{attribute 'linkalways'} 
{attribute 'no_explicit_call' := 'This FB is a CLASS and must be accessed using methods or properties'}
{attribute 'enable_dynamic_creation'}
FUNCTION_BLOCK _ETcVnTimestamp EXTENDS EnumDatatypeBase
VAR
	localData : ETcVnTimestamp;
	activeData : REFERENCE TO ETcVnTimestamp;
	enumBaseDatatype : _ULINT(localData);
END_VAR

METHOD PRIVATE AddLocalEnumeration
VAR_INPUT
	Enumeration : T_MAXSTRING;
	Value : ETcVnTimestamp;
END_VAR
AddEnumeration(Enumeration, Value);
END_METHOD

PROPERTY PUBLIC Address : PVOID
GET
Address := ADR(activeData);
END_GET
END_PROPERTY

METHOD PUBLIC ClearReference
VAR_INPUT
END_VAR
activeData REF= localData;
SetBaseDatatypeReference();
END_METHOD

METHOD PUBLIC Clone : I_Datatype
VAR
    pClone : POINTER TO _ETcVnTimestamp;
END_VAR
pClone := __NEW(_ETcVnTimestamp(InitialValue := Value));
Clone := pClone^;
END_METHOD

METHOD FB_init : BOOL
VAR_INPUT
	bInitRetains : BOOL; // if TRUE, the retain variables are initialized (warm start / cold start)
	bInCopyCode : BOOL;  // if TRUE, the instance afterwards gets moved into the copy code (online change)
	InitialValue : ETcVnTimestamp;
END_VAR
localData := InitialValue;
AddBaseDatatype(enumBaseDatatype);
ClearReference();

AddLocalEnumeration('TCVN_TS_IMAGE_COMPLETED', ETcVnTimestamp.TCVN_TS_IMAGE_COMPLETED);
AddLocalEnumeration('TCVN_TS_RECEPTION_STARTED', ETcVnTimestamp.TCVN_TS_RECEPTION_STARTED);
AddLocalEnumeration('TCVN_TS_RECEPTION_FINISHED', ETcVnTimestamp.TCVN_TS_RECEPTION_FINISHED);
AddLocalEnumeration('TCVN_TS_GETCURRENTIMAGE', ETcVnTimestamp.TCVN_TS_GETCURRENTIMAGE);
AddLocalEnumeration('TCVN_TS_CAMERA', ETcVnTimestamp.TCVN_TS_CAMERA);
AddLocalEnumeration('TCVN_TS_CUSTOM', ETcVnTimestamp.TCVN_TS_CUSTOM);
AddLocalEnumeration('TCVN_TS_LAST_CHANGE', ETcVnTimestamp.TCVN_TS_LAST_CHANGE);
END_METHOD

PROPERTY PUBLIC Identifier : T_MAXSTRING
GET
Identifier := 'ETcVnTimestamp';
END_GET
END_PROPERTY

METHOD IsEnumeratorValueEqual : BOOL
VAR_INPUT
	Enumerator : I_KeyValueForwardEnumerator;
END_VAR
VAR
	storedValue : ETcVnTimestamp;
END_VAR
IF NOT Enumerator.TryGet(storedValue) THEN
	RETURN;
END_IF

IsEnumeratorValueEqual := storedValue = activeData;
END_METHOD

METHOD PUBLIC MakeReferenceTo
VAR_INPUT
	ReferenceTarget : REFERENCE TO ETcVnTimestamp;
END_VAR
activeData REF= ReferenceTarget;
SetBaseDatatypeReference();
END_METHOD

METHOD PROTECTED SetBaseDatatypeReference
VAR_INPUT
END_VAR
enumBaseDatatype.MakeReferenceTo(activeData);
END_METHOD

PROPERTY PUBLIC Size : UDINT
GET
Size := SIZEOF(activeData);
END_GET
END_PROPERTY

METHOD TryMakeReferenceTo : BOOL
VAR_INPUT
	Target : I_Datatype;
END_VAR
VAR
	pTargetData : POINTER TO ETcVnTimestamp;
END_VAR
IF NOT IsEquivalentTo(Target) THEN
	RETURN;
END_IF

pTargetData := Target.Address;
activeData REF= pTargetData^;
SetBaseDatatypeReference();
TryMakeReferenceTo := TRUE;
END_METHOD

PROPERTY PUBLIC Value : ETcVnTimestamp
GET
Value := activeData;
END_GET
SET
activeData := Value;
END_SET
END_PROPERTY

END_FUNCTION_BLOCK

(* stored: Version 1.1.0.1, ProductVersion 3.1.4024.13
   POU _ETcVnTimestamp: Id {d310adf1-2d37-00bd-1115-27d104ed3ef1}, SpecialFunc None
   Folder Core: Id {77af2560-cced-0daa-1211-123cfc3f2b65}
   Folder Protected: Id {f197ed99-828c-03bc-1837-1248521862bf}
   Folder Customize: Id {a26a2583-c016-0ec1-1b4d-be17805a6222}
   Folder Constructor: Id {2f2e0018-e3d4-06bb-102f-a67267979187}
   Folder Private: Id {c1d5397d-7f83-04fc-00f1-6b2625b52d99}
   Folder Protected: Id {52aaf5b4-eb11-0bc2-3716-f2f8b90090b1}
   Method AddLocalEnumeration: Id {77d22b0d-a8d9-0cc2-2753-4dd5ac642356}
   Property Address: Id {859ab322-5f62-0381-1503-fb6a93686b75}
   Get Get: Id {3d2bfc6b-7a64-08f3-1a17-af947191ef54}
   Method ClearReference: Id {95f88eef-d490-0511-0202-d3cf57e680b4}
   Method Clone: Id {daa1e185-a8b6-0b39-333e-ce61777f51c2}
   Method FB_init: Id {9f033ef3-530e-0765-08c7-8923a6e6ad97}
   Property Identifier: Id {06515588-f3ce-01c0-170e-fa8c1bf802a9}
   Get Get: Id {703d6092-be97-00bd-3087-38ab1f5f081f}
   Method IsEnumeratorValueEqual: Id {560050ac-7653-0d30-00f8-a6d25b695e98}
   Method MakeReferenceTo: Id {61668270-db79-04e9-0e90-5eb69891bd84}
   Method SetBaseDatatypeReference: Id {a930ae43-7be7-0941-2b36-9713d6b68d23}
   Property Size: Id {703e7216-26af-0e76-129d-cd275b9226dd}
   Get Get: Id {b1278cfc-cac0-06f6-1403-98d4a5db3bc7}
   Method TryMakeReferenceTo: Id {b6418bcc-2ce6-07bf-3e40-2e47a18b59e6}
   Property Value: Id {7f9bfb73-92b5-0ca9-1500-7675d08efd7d}
   Get Get: Id {dd694c81-71d0-076b-2539-de2f718b5b9c}
   Set Set: Id {6d461b41-5e23-0582-2186-95984b105a00} *)
